// TwinCAT 3 PLC project PLC2
// ProgramVersion: 3.1.4026.23
// libraries:
//   Tc2_EtherCAT, * (Beckhoff Automation GmbH)
//   Tc2_Standard, * (Beckhoff Automation GmbH)
//   Tc2_System, * (Beckhoff Automation GmbH)
// project tree:
//   / Plc2Task.TcTTO
//   POUs/ F_ConsumeTime.TcPOU, PRG_PLC2.TcPOU
// (motion and I/O tree: see PLC project plc1)
// real-time tasks:
//   TASK Plc1Task: cycle T#10ms, priority 10, ADS port 350
//   TASK Plc2Task: cycle T#10ms, priority 14, ADS port 351
//   TASK EcSlaveTask: cycle T#10ms, priority 3, ADS port 352
// variable links:

CONFIGURATION PLC2
    RESOURCE PLC ON TwinCAT3
        TASK Plc2Task(INTERVAL := T#10ms, PRIORITY := 14);
        PROGRAM PRG_PLC2 WITH Plc2Task : PRG_PLC2;
    END_RESOURCE
END_CONFIGURATION

// ---- POUs/PRG_PLC2.TcPOU
PROGRAM PRG_PLC2
VAR
	EncoderValue AT %I* : UINT;
	Pos					: LREAL;
END_VAR

F_ConsumeTime(20);

Pos:= UINT_TO_LREAL(EncoderValue)*100;

END_PROGRAM

// ---- POUs/F_ConsumeTime.TcPOU
FUNCTION F_ConsumeTime
VAR_INPUT
	Us		:UDINT;
END_VAR
VAR
		tCurr, tEnd : T_DCTIME64;
END_VAR

tCurr := F_GetActualDcTime64();
tEnd  := tCurr + (Us * EC_DCTIME_TICKSPERMSEC64 / 1000);
WHILE (tCurr < tEnd) DO
	tCurr := F_GetActualDcTime64();
END_WHILE

END_FUNCTION
